PROGRAM Mission
VAR
	Mission1: BOOL;
	Mission2: BOOL;
	NoMission: BOOL;
	AutoRunning: BOOL;
	Mission1Start: BOOL;
	Mission1Done: BOOL;
	Mission2Start: BOOL;
	Mission2Done: BOOL;
END_VAR

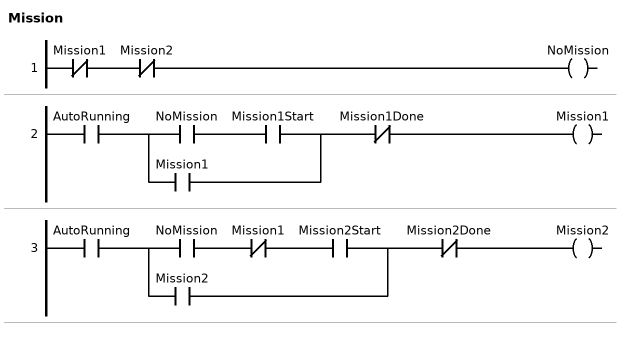
// NETWORK 1
NoMission := NOT Mission1 AND NOT Mission2;

// NETWORK 2
Mission1 := AutoRunning AND (NoMission AND Mission1Start OR Mission1) AND NOT Mission1Done;

// NETWORK 3
Mission2 := AutoRunning AND (NoMission AND NOT Mission1 AND Mission2Start OR Mission2) AND NOT Mission2Done;

END_PROGRAM

(* stored: Version 1.1.0.1, ProductVersion 3.1.4024.10
   POU Mission: Id {a3bb4db7-32ef-4dcf-b066-28622cc60419}, SpecialFunc None *)
